// TIA Portal V16 export
// export: Created 2024-09-05T17:39:23.7110622Z, ExportSetting WithDefaults, DisplayName Totally Integrated Automation Portal, DisplayVersion V16 Update 6, DisplayName TIA Portal Version Control Interface, DisplayVersion V16 Update 2, DisplayName TIA Portal Openness, DisplayVersion V16 Update 6, DisplayName STEP 7 Professional, DisplayVersion V16 Update 6, DisplayName STEP 7 Safety, DisplayVersion V16, DisplayName WinCC Advanced, DisplayVersion V16 Update 6
DATA_BLOCK "DB_IJCoreMain"   // DB1000
VERSION : 0.1
// stored: AutoNumber false, DBAccessibleFromOPCUA true, InstanceOfName IJCoreMain, InstanceOfType FB
"IJCoreMain"
   // VAR
   //    Enable : Bool := true;
   //    Mode : UInt := 1;
   //    Indicator : Int;
   //    AlarmReset : Bool;
   //    AWAKE_SIGNAL { S7_SetPoint := 'True'} : "AWAKE_SIGNAL";
   //    MSG : Array[1..20] of "IJCoreMessageProcotol";
   //    NFP { S7_SetPoint := 'True'} : Array[1..4] of String[30];
   // END_VAR
BEGIN
END_DATA_BLOCK
